TYPE st_Event :
STRUCT
	e_Event_Type : e_Event_Type;
	e_Event_Severity : TcEventSeverity;
	n_Event_Identity : UDINT;
	s_Event_Text : STRING(255);
	dt_Timestamp : DATE_AND_TIME;
END_STRUCT
END_TYPE

(* stored: Version 1.1.0.1
   DUT st_Event: Id {40a63048-541b-46ea-b8e8-913401d4b898} *)
